// Mitsubishi GX Works2 project: 230929-001- exercicios de hoje   PLC: Q03UDV

// task Task_01 (event TRUE, interval 0, priority 31): POU_01

PROGRAM POU_01
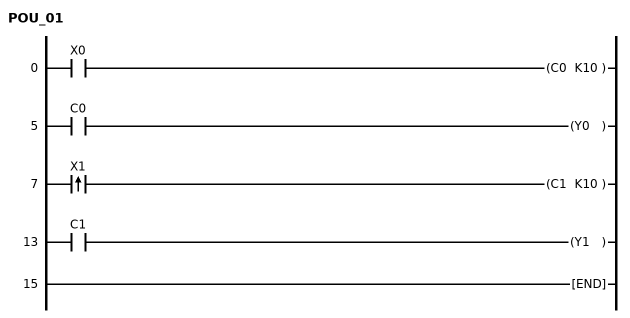
0     LD      X0
      OUT     C0 K10
5     LD      C0
      OUT     Y0
7     LDP     X1
      OUT     C1 K10
13    LD      C1
      OUT     Y1
15    END
END_PROGRAM
